TYPE ST_TsConnectionInfoEP1957 :
(*******************************************************************************************************
Description			:	Connection information data of EtherCAT Slaves with 2 byte input and 2 byte output safe data  
Supported terminals : 	EP1957
Date 				:	04.11.2018
********************************************************************************************************)
STRUCT

	nState  								:USINT;
	nDiag 	 								:USINT;
	nInOutSafeDataByte1						:BYTE;
	nInOutSafeDataByte2						:BYTE;
	nInOutSafeDataByte3						:BYTE;
	nInOutSafeDataByte4						:BYTE;

END_STRUCT
END_TYPE
(* End *)

(* stored: Version 1.1.0.1, ProductVersion 3.1.4022.16
   DUT ST_TsConnectionInfoEP1957: Id {89bad86b-74e4-4823-a33b-106e95176b08} *)
